  994 = 'S6_Prompts Default 994' | German: 'S6_Prompts German 994' | French: 'S6_Prompts French 994'
  995 = 'S6_Prompts Default 995' | German: 'S6_Prompts German 995' | French: 'S6_Prompts French 995'
  996 = 'S6_Prompts Default 996' | German: 'S6_Prompts German 996' | French: 'S6_Prompts French 996'
  997 = 'S6_Prompts Default 997' | German: 'S6_Prompts German 997' | French: 'S6_Prompts French 997'
  998 = 'S6_Prompts Default 998' | German: 'S6_Prompts German 998' | French: 'S6_Prompts French 998'
  999 = 'S6_Prompts Default 999' | German: 'S6_Prompts German 999' | French: 'S6_Prompts French 999'
  1000 = 'S6_Prompts Default 1000' | German: 'S6_Prompts German 1000' | French: 'S6_Prompts French 1000'
   = ''
END_TEXTLIST

(* stored: Version 1.1.0.1, ProductVersion 3.1.4024.12
   TextList S6_Prompts: Id {4fc238e8-9672-434e-9510-75cf3fdb9018} *)
